Universal Robots PolyScope program: fun3.urp

Program fun3 (installation=default directory=/programs createdIn=5.9.1.1031110 lastSavedIn=5.9.1.1031110 robotSerialNumber=20195501059)
Calibrated DH parameters: a=[0.000146, -0.418764, -0.053981, 0.000058, -0.000023, 0]; d=[0.162545, 37.319448, -206.067439, 168.881546, 0.09955, 0.099464]; alpha=[1.57004, -0.001979, 0.002304, 1.570607, -1.57066, 0]; deltaTheta=[0, -0.174616, -1.258233, 1.432844, -0.000001, 0]
Robot Program (runOnlyOnce=true)
  MoveJ speed 60 deg/s, acceleration 80 deg/s^2 (useActiveTCP=true) feature=Base
    Waypoint Waypoint_1: TCP in base x=107.141 y=-470.469 z=45.786 mm, rx=-2.748 ry=-1.5225 rz=0 rad; joints [86.741, -80.237, 122.137, -131.89, 270.055, -241.197] deg; TCP offset x=0 y=0 z=174 mm, rx=0 ry=0 rz=0 rad
  MoveL speed 250 mm/s, acceleration 1200 mm/s^2 (useActiveTCP=true) feature=Base
    Waypoint Waypoint_2: TCP in base x=250.856 y=-349.536 z=45.806 mm, rx=-2.748 ry=-1.5224 rz=0.0001 rad; joints [107.569, -86.969, 129.96, -132.982, 270.071, -220.363] deg
  URCap Olis Teleop (Olis Teleop, Olis Robotics) dataModel(OperatorMessage=Teleoperation demo time!)
  MoveL speed 250 mm/s, acceleration 1200 mm/s^2 (useActiveTCP=true) feature=Base
    Waypoint Waypoint_1: TCP in base x=107.141 y=-470.469 z=45.786 mm, rx=-2.748 ry=-1.5225 rz=0 rad; joints [86.741, -80.237, 122.137, -131.89, 270.055, -241.197] deg
